(* CODESYS project bibliothek_2.library
   Company: Viessmann
   Title: GWP_Libary_Visu_2
   Placeholder: GWP_Libary_Visu_2
   Version: 0.0.1

Project tree, tasks and I/O mapping:
  libraries: Tc2_Standard, * (Beckhoff Automation GmbH); Tc2_System, * (Beckhoff Automation GmbH); Tc3_Module, * (Beckhoff Automation GmbH)
  DUTs/
  GVLs/
  POUs/
    program MAIN [ST]
  Version/
    global variables Global_Version
  VISUs/
    Sollwerte/
      visualisation Sollwerte_Test
    image pool Icon
  00000000-0000-0000-0000-000000000000|C:\Users\kuzr\Documents\Visual Studio 2013\Bildersammlung_VI\IC_102000\energietraeger_biomasse_fehler.png
  00000000-0000-0000-0000-000000000000|C:\Users\kuzr\Documents\Visual Studio 2013\Bildersammlung_VI\IC_102000\energietraeger_biomasse_inaktiv.png
  00000000-0000-0000-0000-000000000000|C:\Users\kuzr\Documents\Visual Studio 2013\Bildersammlung_VI\IC_102000\energietraeger_gas.png
  00000000-0000-0000-0000-000000000000|C:\Users\kuzr\Documents\Visual Studio 2013\Bildersammlung_VI\IC_102000\energietraeger_gas_fehler.png
  00000000-0000-0000-0000-000000000000|C:\Users\kuzr\Documents\Visual Studio 2013\Bildersammlung_VI\IC_102000\energietraeger_naturwaerme.png
  00000000-0000-0000-0000-000000000000|C:\Users\kuzr\Documents\Visual Studio 2013\Bildersammlung_VI\IC_102000\energietraeger_naturwaerme_fehler (2).png
  00000000-0000-0000-0000-000000000000|C:\Users\kuzr\Documents\Visual Studio 2013\Bildersammlung_VI\IC_102000\energietraeger_naturwaerme_fehler.png
  00000000-0000-0000-0000-000000000000|C:\Users\kuzr\Documents\Visual Studio 2013\Bildersammlung_VI\IC_102000\energietraeger_naturwaerme_inaktiv.png
  00000000-0000-0000-0000-000000000000|C:\Users\kuzr\Documents\Visual Studio 2013\Bildersammlung_VI\IC_102000\energietraeger_oel.png
  00000000-0000-0000-0000-000000000000|C:\Users\kuzr\Documents\Visual Studio 2013\Bildersammlung_VI\IC_102000\energietraeger_oel_inaktiv.png
  00000000-0000-0000-0000-000000000000|C:\Users\kuzr\Documents\Visual Studio 2013\Bildersammlung_VI\IC_102000\heizkreis_direkt (2).png
  00000000-0000-0000-0000-000000000000|C:\Users\kuzr\Documents\Visual Studio 2013\Bildersammlung_VI\IC_102000\heizkreis_direkt.png
  00000000-0000-0000-0000-000000000000|C:\Users\kuzr\Documents\Visual Studio 2013\Bildersammlung_VI\IC_102000\heizkreis_direkt_fehler.png
  00000000-0000-0000-0000-000000000000|C:\Users\kuzr\Documents\Visual Studio 2013\Bildersammlung_VI\IC_102000\heizkreis_direkt_inaktiv (2).png
  00000000-0000-0000-0000-000000000000|C:\Users\kuzr\Documents\Visual Studio 2013\Bildersammlung_VI\IC_102000\heizkreis_direkt_inaktiv.png
  00000000-0000-0000-0000-000000000000|C:\Users\kuzr\Documents\Visual Studio 2013\Bildersammlung_VI\IC_102000\heizkreis_fussbodenheizung.png
  00000000-0000-0000-0000-000000000000|C:\Users\kuzr\Documents\Visual Studio 2013\Bildersammlung_VI\IC_102000\heizkreis_fussbodenheizung_fehler.png
  00000000-0000-0000-0000-000000000000|C:\Users\kuzr\Documents\Visual Studio 2013\Bildersammlung_VI\IC_102000\heizkreis_fussbodenheizung_inaktiv.png
  00000000-0000-0000-0000-000000000000|C:\Users\kuzr\Documents\Visual Studio 2013\Bildersammlung_VI\IC_102000\heizkreis_mischer.png
  00000000-0000-0000-0000-000000000000|C:\Users\kuzr\Documents\Visual Studio 2013\Bildersammlung_VI\IC_102000\heizkreis_mischer_fehler.png
  00000000-0000-0000-0000-000000000000|C:\Users\kuzr\Documents\Visual Studio 2013\Bildersammlung_VI\IC_102000\heizkreis_mischer_inaktiv.png
  00000000-0000-0000-0000-000000000000|C:\Users\kuzr\Documents\Visual Studio 2013\Bildersammlung_VI\IC_102000\IC_102015_klappen_02.png
  00000000-0000-0000-0000-000000000000|C:\Users\kuzr\Documents\Visual Studio 2013\Bildersammlung_VI\IC_102000\klappen_01 (2).png
  00000000-0000-0000-0000-000000000000|C:\Users\kuzr\Documents\Visual Studio 2013\Bildersammlung_VI\IC_102000\klappen_01.png
  00000000-0000-0000-0000-000000000000|C:\Users\kuzr\Documents\Visual Studio 2013\Bildersammlung_VI\IC_102000\klappen_02.png
  00000000-0000-0000-0000-000000000000|C:\Users\kuzr\Documents\Visual Studio 2013\Bildersammlung_VI\IC_102000\komponente_detail_heizkreis.png
  00000000-0000-0000-0000-000000000000|C:\Users\kuzr\Documents\Visual Studio 2013\Bildersammlung_VI\IC_102000\komponente_detail_klappe (2).png
  00000000-0000-0000-0000-000000000000|C:\Users\kuzr\Documents\Visual Studio 2013\Bildersammlung_VI\IC_102000\komponente_detail_klappe.png
  00000000-0000-0000-0000-000000000000|C:\Users\kuzr\Documents\Visual Studio 2013\Bildersammlung_VI\IC_102000\komponente_detail_klappe_fehler (2).png
  00000000-0000-0000-0000-000000000000|C:\Users\kuzr\Documents\Visual Studio 2013\Bildersammlung_VI\IC_102000\komponente_detail_klappe_fehler.png
  00000000-0000-0000-0000-000000000000|C:\Users\kuzr\Documents\Visual Studio 2013\Bildersammlung_VI\IC_102000\komponente_detail_klappe_inaktiv.png
  00000000-0000-0000-0000-000000000000|C:\Users\kuzr\Documents\Visual Studio 2013\Bildersammlung_VI\IC_102000\komponente_detail_klappe_inaktiv_2.png
  00000000-0000-0000-0000-000000000000|C:\Users\kuzr\Documents\Visual Studio 2013\Bildersammlung_VI\IC_102000\komponente_detail_mischer_01.png
  00000000-0000-0000-0000-000000000000|C:\Users\kuzr\Documents\Visual Studio 2013\Bildersammlung_VI\IC_102000\komponente_detail_mischer_02.png
  00000000-0000-0000-0000-000000000000|C:\Users\kuzr\Documents\Visual Studio 2013\Bildersammlung_VI\IC_102000\komponente_detail_mischer_fehler.png
  00000000-0000-0000-0000-000000000000|C:\Users\kuzr\Documents\Visual Studio 2013\Bildersammlung_VI\IC_102000\komponente_detail_mischer_inaktiv.png
  00000000-0000-0000-0000-000000000000|C:\Users\kuzr\Documents\Visual Studio 2013\Bildersammlung_VI\IC_102000\komponente_detail_pumpe.png
  00000000-0000-0000-0000-000000000000|C:\Users\kuzr\Documents\Visual Studio 2013\Bildersammlung_VI\IC_102000\komponente_detail_pumpe_fehler.png
  00000000-0000-0000-0000-000000000000|C:\Users\kuzr\Documents\Visual Studio 2013\Bildersammlung_VI\IC_102000\komponente_detail_pumpe_inaktiv.png
  00000000-0000-0000-0000-000000000000|C:\Users\kuzr\Documents\Visual Studio 2013\Bildersammlung_VI\IC_102000\mischer_01.png
  00000000-0000-0000-0000-000000000000|C:\Users\kuzr\Documents\Visual Studio 2013\Bildersammlung_VI\IC_102000\mischer_02.png
  00000000-0000-0000-0000-000000000000|C:\Users\kuzr\Documents\Visual Studio 2013\Bildersammlung_VI\IC_102000\mischer_03.png
  00000000-0000-0000-0000-000000000000|C:\Users\kuzr\Documents\Visual Studio 2013\Bildersammlung_VI\IC_102000\mischer_04.png
  00000000-0000-0000-0000-000000000000|C:\Users\kuzr\Documents\Visual Studio 2013\Bildersammlung_VI\IC_102000\mischer_05.png
  00000000-0000-0000-0000-000000000000|C:\Users\kuzr\Documents\Visual Studio 2013\Bildersammlung_VI\IC_102000\mischer_06.png
  00000000-0000-0000-0000-000000000000|C:\Users\kuzr\Documents\Visual Studio 2013\Bildersammlung_VI\IC_102000\mischer_07.png
  00000000-0000-0000-0000-000000000000|C:\Users\kuzr\Documents\Visual Studio 2013\Bildersammlung_VI\IC_102000\mischer_08.png
  00000000-0000-0000-0000-000000000000|C:\Users\kuzr\Documents\Visual Studio 2013\Bildersammlung_VI\IC_102000\mischer_09.png
  00000000-0000-0000-0000-000000000000|C:\Users\kuzr\Documents\Visual Studio 2013\Bildersammlung_VI\IC_102000\mischer_10.png
  00000000-0000-0000-0000-000000000000|C:\Users\kuzr\Documents\Visual Studio 2013\Bildersammlung_VI\IC_102000\mischer_11.png
  00000000-0000-0000-0000-000000000000|C:\Users\kuzr\Documents\Visual Studio 2013\Bildersammlung_VI\IC_102000\mischer_12.png
  00000000-0000-0000-0000-000000000000|C:\Users\kuzr\Documents\Visual Studio 2013\Bildersammlung_VI\IC_102000\pumpe_links.png
  00000000-0000-0000-0000-000000000000|C:\Users\kuzr\Documents\Visual Studio 2013\Bildersammlung_VI\IC_102000\pumpe_oben.png
  00000000-0000-0000-0000-000000000000|C:\Users\kuzr\Documents\Visual Studio 2013\Bildersammlung_VI\IC_102000\pumpe_rechts.png
  00000000-0000-0000-0000-000000000000|C:\Users\kuzr\Documents\Visual Studio 2013\Bildersammlung_VI\IC_102000\pumpe_unten.png
  00000000-0000-0000-0000-000000000000|C:\Users\kuzr\Documents\Visual Studio 2013\Bildersammlung_VI\IC_102000\speicher_eis.png
  00000000-0000-0000-0000-000000000000|C:\Users\kuzr\Documents\Visual Studio 2013\Bildersammlung_VI\IC_102000\speicher_eis_fehler.png
  00000000-0000-0000-0000-000000000000|C:\Users\kuzr\Documents\Visual Studio 2013\Bildersammlung_VI\IC_102000\speicher_eis_inaktiv.png
  00000000-0000-0000-0000-000000000000|C:\Users\kuzr\Documents\Visual Studio 2013\Bildersammlung_VI\IC_102000\speicher_heizen.png
  00000000-0000-0000-0000-000000000000|C:\Users\kuzr\Documents\Visual Studio 2013\Bildersammlung_VI\IC_102000\speicher_heizen_fehler.png
  00000000-0000-0000-0000-000000000000|C:\Users\kuzr\Documents\Visual Studio 2013\Bildersammlung_VI\IC_102000\speicher_heizen_inaktiv.png
  00000000-0000-0000-0000-000000000000|C:\Users\kuzr\Documents\Visual Studio 2013\Bildersammlung_VI\IC_102000\speicher_warmwasser.png
  00000000-0000-0000-0000-000000000000|C:\Users\kuzr\Documents\Visual Studio 2013\Bildersammlung_VI\IC_102000\speicher_warmwasser_fehler.png
  00000000-0000-0000-0000-000000000000|C:\Users\kuzr\Documents\Visual Studio 2013\Bildersammlung_VI\IC_102000\speicher_warmwasser_inaktiv.png
  00000000-0000-0000-0000-000000000000|C:\Users\kuzr\Documents\Visual Studio 2013\Bildersammlung_VI\IC_102000\energietraeger_biomasse.png
  00000000-0000-0000-0000-000000000000|C:\Users\kuzr\Documents\Visual Studio 2013\Bildersammlung_VI\IC_106000\komponente_brenner.png
  00000000-0000-0000-0000-000000000000|C:\Users\kuzr\Documents\Visual Studio 2013\Bildersammlung_VI\IC_106000\komponente_brenner_fehler.png
  00000000-0000-0000-0000-000000000000|C:\Users\kuzr\Documents\Visual Studio 2013\Bildersammlung_VI\IC_106000\komponente_brenner_inaktiv.png
  00000000-0000-0000-0000-000000000000|C:\Users\kuzr\Documents\Visual Studio 2013\Bildersammlung_VI\IC_106000\speicher.png
  00000000-0000-0000-0000-000000000000|C:\Users\kuzr\Documents\Visual Studio 2013\Bildersammlung_VI\IC_106000\speicher_eis.png
  00000000-0000-0000-0000-000000000000|C:\Users\kuzr\Documents\Visual Studio 2013\Bildersammlung_VI\IC_106000\system_leistung_nicht_touchbar.png
  00000000-0000-0000-0000-000000000000|C:\Users\kuzr\Documents\Visual Studio 2013\Bildersammlung_VI\IC_106000\system_leistung_touchbar.png
  00000000-0000-0000-0000-000000000000|C:\Users\kuzr\Documents\Visual Studio 2013\Bildersammlung_VI\IC_106000\waermetauscher.png
  00000000-0000-0000-0000-000000000000|C:\Users\kuzr\Documents\Visual Studio 2013\Bildersammlung_VI\IC_106000\weiche.png
  00000000-0000-0000-0000-000000000000|C:\Users\kuzr\Documents\Visual Studio 2013\Bildersammlung_VI\IC_108000\komponente_brenner_fehler.png
  00000000-0000-0000-0000-000000000000|C:\Users\kuzr\Documents\Visual Studio 2013\Bildersammlung_VI\IC_108000\komponente_brenner_inaktiv.png
  00000000-0000-0000-0000-000000000000|C:\Users\kuzr\Documents\Visual Studio 2013\Bildersammlung_VI\IC_108000\speicher.png
  00000000-0000-0000-0000-000000000000|C:\Users\kuzr\Documents\Visual Studio 2013\Bildersammlung_VI\IC_108000\speicher_eis.png
  00000000-0000-0000-0000-000000000000|C:\Users\kuzr\Documents\Visual Studio 2013\Bildersammlung_VI\IC_108000\komponente_brenner.png
  00000000-0000-0000-0000-000000000000|C:\Users\kuzr\Documents\Visual Studio 2013\Bildersammlung_VI\IC_111000\bildschirm_reinigen.png
  00000000-0000-0000-0000-000000000000|C:\Users\kuzr\Documents\Visual Studio 2013\Bildersammlung_VI\IC_111000\dokumentation.png
  00000000-0000-0000-0000-000000000000|C:\Users\kuzr\Documents\Visual Studio 2013\Bildersammlung_VI\IC_111000\kontaktdaten_nutzer.png
  00000000-0000-0000-0000-000000000000|C:\Users\kuzr\Documents\Visual Studio 2013\Bildersammlung_VI\IC_111000\kontaktdaten_viessmann.png
  00000000-0000-0000-0000-000000000000|C:\Users\kuzr\Documents\Visual Studio 2013\Bildersammlung_VI\IC_111000\nutzeranmeldung.png
  00000000-0000-0000-0000-000000000000|C:\Users\kuzr\Documents\Visual Studio 2013\Bildersammlung_VI\IC_111000\oberflaeche_schließen.png
  00000000-0000-0000-0000-000000000000|C:\Users\kuzr\Documents\Visual Studio 2013\Bildersammlung_VI\IC_111000\pruefbetrieb.png
  00000000-0000-0000-0000-000000000000|C:\Users\kuzr\Documents\Visual Studio 2013\Bildersammlung_VI\IC_111000\system_konfigurieren.png
  00000000-0000-0000-0000-000000000000|C:\Users\kuzr\Documents\Visual Studio 2013\Bildersammlung_VI\IC_111000\betriebszaehler_zuruecksetzen.png
  00000000-0000-0000-0000-000000000000|C:\Users\kuzr\Documents\Visual Studio 2013\Bildersammlung_VI\IC_112000\abschaltbetrieb.png
  00000000-0000-0000-0000-000000000000|C:\Users\kuzr\Documents\Visual Studio 2013\Bildersammlung_VI\IC_112000\aktiv.png
  00000000-0000-0000-0000-000000000000|C:\Users\kuzr\Documents\Visual Studio 2013\Bildersammlung_VI\IC_112000\an.png
  00000000-0000-0000-0000-000000000000|C:\Users\kuzr\Documents\Visual Studio 2013\Bildersammlung_VI\IC_112000\astatur_01.png
  00000000-0000-0000-0000-000000000000|C:\Users\kuzr\Documents\Visual Studio 2013\Bildersammlung_VI\IC_112000\auf.png
  00000000-0000-0000-0000-000000000000|C:\Users\kuzr\Documents\Visual Studio 2013\Bildersammlung_VI\IC_112000\aus.png
  00000000-0000-0000-0000-000000000000|C:\Users\kuzr\Documents\Visual Studio 2013\Bildersammlung_VI\IC_112000\bedingung_erfuellt.png
  00000000-0000-0000-0000-000000000000|C:\Users\kuzr\Documents\Visual Studio 2013\Bildersammlung_VI\IC_112000\bedingung_nicht_erfuellt.png
  00000000-0000-0000-0000-000000000000|C:\Users\kuzr\Documents\Visual Studio 2013\Bildersammlung_VI\IC_112000\email_prueftaste.png
  00000000-0000-0000-0000-000000000000|C:\Users\kuzr\Documents\Visual Studio 2013\Bildersammlung_VI\IC_112000\erfuellt.png
  00000000-0000-0000-0000-000000000000|C:\Users\kuzr\Documents\Visual Studio 2013\Bildersammlung_VI\IC_112000\exportieren.png
  00000000-0000-0000-0000-000000000000|C:\Users\kuzr\Documents\Visual Studio 2013\Bildersammlung_VI\IC_112000\frostschutzbetrieb.png
  00000000-0000-0000-0000-000000000000|C:\Users\kuzr\Documents\Visual Studio 2013\Bildersammlung_VI\IC_112000\haeckchen_ungesetzt (2).png
  00000000-0000-0000-0000-000000000000|C:\Users\kuzr\Documents\Visual Studio 2013\Bildersammlung_VI\IC_112000\haeckchen_ungesetzt.png
  00000000-0000-0000-0000-000000000000|C:\Users\kuzr\Documents\Visual Studio 2013\Bildersammlung_VI\IC_112000\home.png
  00000000-0000-0000-0000-000000000000|C:\Users\kuzr\Documents\Visual Studio 2013\Bildersammlung_VI\IC_112000\home_uebersicht.png
  00000000-0000-0000-0000-000000000000|C:\Users\kuzr\Documents\Visual Studio 2013\Bildersammlung_VI\IC_112000\inaktiv.png
  00000000-0000-0000-0000-000000000000|C:\Users\kuzr\Documents\Visual Studio 2013\Bildersammlung_VI\IC_112000\intervall.png
  00000000-0000-0000-0000-000000000000|C:\Users\kuzr\Documents\Visual Studio 2013\Bildersammlung_VI\IC_112000\Itastatur_03.png
  00000000-0000-0000-0000-000000000000|C:\Users\kuzr\Documents\Visual Studio 2013\Bildersammlung_VI\IC_112000\ja.png
  00000000-0000-0000-0000-000000000000|C:\Users\kuzr\Documents\Visual Studio 2013\Bildersammlung_VI\IC_112000\kopieren.png
  00000000-0000-0000-0000-000000000000|C:\Users\kuzr\Documents\Visual Studio 2013\Bildersammlung_VI\IC_112000\laden.png
  00000000-0000-0000-0000-000000000000|C:\Users\kuzr\Documents\Visual Studio 2013\Bildersammlung_VI\IC_112000\listenansicht.png
  00000000-0000-0000-0000-000000000000|C:\Users\kuzr\Documents\Visual Studio 2013\Bildersammlung_VI\IC_112000\meldelisten_archiv.png
  00000000-0000-0000-0000-000000000000|C:\Users\kuzr\Documents\Visual Studio 2013\Bildersammlung_VI\IC_112000\meldelisten_einstellungen.png
  00000000-0000-0000-0000-000000000000|C:\Users\kuzr\Documents\Visual Studio 2013\Bildersammlung_VI\IC_112000\meldungen_weiterleiten.png
  00000000-0000-0000-0000-000000000000|C:\Users\kuzr\Documents\Visual Studio 2013\Bildersammlung_VI\IC_112000\menue.png
  00000000-0000-0000-0000-000000000000|C:\Users\kuzr\Documents\Visual Studio 2013\Bildersammlung_VI\IC_112000\minus.png
  00000000-0000-0000-0000-000000000000|C:\Users\kuzr\Documents\Visual Studio 2013\Bildersammlung_VI\IC_112000\nein.png
  00000000-0000-0000-0000-000000000000|C:\Users\kuzr\Documents\Visual Studio 2013\Bildersammlung_VI\IC_112000\nicht_erfuellt.png
  00000000-0000-0000-0000-000000000000|C:\Users\kuzr\Documents\Visual Studio 2013\Bildersammlung_VI\IC_112000\normalbetrieb.png
  00000000-0000-0000-0000-000000000000|C:\Users\kuzr\Documents\Visual Studio 2013\Bildersammlung_VI\IC_112000\pfeil_rechts.png
  00000000-0000-0000-0000-000000000000|C:\Users\kuzr\Documents\Visual Studio 2013\Bildersammlung_VI\IC_112000\plus.png
  00000000-0000-0000-0000-000000000000|C:\Users\kuzr\Documents\Visual Studio 2013\Bildersammlung_VI\IC_112000\quittieren_aus.png
  00000000-0000-0000-0000-000000000000|C:\Users\kuzr\Documents\Visual Studio 2013\Bildersammlung_VI\IC_112000\quittierena_an.png
  00000000-0000-0000-0000-000000000000|C:\Users\kuzr\Documents\Visual Studio 2013\Bildersammlung_VI\IC_112000\radiobutton_gesetzt.png
  00000000-0000-0000-0000-000000000000|C:\Users\kuzr\Documents\Visual Studio 2013\Bildersammlung_VI\IC_112000\radiobutton_ungesetzt.png
  text list GlobalTextList
*)

// Version/Global_Version
{attribute 'TcGenerated'}
// This function has been automatically generated from the project information.
VAR_GLOBAL CONSTANT
	{attribute 'const_non_replaced'}
	{attribute 'linkalways'}
	stLibVersion_GWP_Libary_Visu_2 : ST_LibVersion := (iMajor := 0, iMinor := 0, iBuild := 1, iRevision := 0, sVersion := '0.0.1');
END_VAR

// POUs/MAIN
PROGRAM MAIN
VAR
END_VAR

END_PROGRAM

// VISUs/Sollwerte/Sollwerte_Test
VISUALIZATION Sollwerte_Test  // 2x2
END_VISUALIZATION
